LIN {X 0,Y 102.749,Z 789.468,A -85,B 0,C 180,E1 -26714.124,E2 -26714.124} C_VEL
LIN {X 0,Y 103.619,Z 785.992,A -85,B 0,C 180,E1 -26722.206,E2 -26722.206} C_VEL
LIN {X 0,Y 105.515,Z 782.796,A -85,B 0,C 180,E1 -26727.611,E2 -26727.611} C_VEL
LIN {X 0,Y 106.613,Z 781.059,A -85,B 0,C 180,E1 -26730.002,E2 -26730.002} C_VEL
LIN {X 0,Y 107.479,Z 777.383,A -85,B 0,C 180,E1 -26733.751,E2 -26733.751} C_VEL
LIN {X 0,Y 105.034,Z 782.053,A -85,B 0,C 180,E1 -26741.582,E2 -26741.582} C_VEL
LIN {X 0,Y 105.176,Z 785.938,A -85,B 0,C 180,E1 -26750.687,E2 -26750.687} C_VEL
LIN {X 0,Y 107.342,Z 787.959,A -85,B 0,C 180,E1 -26757.28,E2 -26757.28} C_VEL
LIN {X 0,Y 112.126,Z 789.61,A -85,B 0,C 180,E1 -26764.343,E2 -26764.343} C_VEL
LIN {X 0,Y 118.966,Z 790.415,A -85,B 0,C 180,E1 -26770.532,E2 -26770.532} C_VEL
LIN {X 0,Y 127.429,Z 790.46,A -85,B 0,C 180,E1 -26775.808,E2 -26775.808} C_VEL
LIN {X 0,Y 137.179,Z 789.707,A -85,B 0,C 180,E1 -26780.22,E2 -26780.22} C_VEL
LIN {X 0,Y 138.04,Z 789.191,A -85,B 0,C 180,E1 -26781.434,E2 -26781.434} C_VEL
LIN {X 0,Y 129.834,Z 786.499,A -85,B 0,C 180,E1 -26785.251,E2 -26785.251} C_VEL
LIN {X 0,Y 125.752,Z 785.046,A -85,B 0,C 180,E1 -26787.045,E2 -26787.045} C_VEL
LIN {X 0,Y 118.099,Z 782.22,A -85,B 0,C 180,E1 -26789.693,E2 -26789.693} C_VEL
LIN {X 0,Y 110.921,Z 778.802,A -85,B 0,C 180,E1 -26792.656,E2 -26792.656} C_VEL
LIN {X 0,Y 107.697,Z 776.475,A -85,B 0,C 180,E1 -26794.945,E2 -26794.945} C_VEL
LIN {X 0,Y 101.788,Z 769.899,A -85,B 0,C 180,E1 -26801.896,E2 -26801.896} C_VEL
LIN {X 0,Y 97.245,Z 760.94,A -85,B 0,C 180,E1 -26810.64,E2 -26810.64} C_VEL
LIN {X 0,Y 94.988,Z 751.352,A -85,B 0,C 180,E1 -26818.938,E2 -26818.938} C_VEL
LIN {X 0,Y 94.512,Z 741.434,A -85,B 0,C 180,E1 -26826.402,E2 -26826.402} C_VEL
LIN {X 0,Y 94.977,Z 731.323,A -85,B 0,C 180,E1 -26832.824,E2 -26832.824} C_VEL
LIN {X 0,Y 96.352,Z 718.316,A -85,B 0,C 180,E1 -26839.712,E2 -26839.712} C_VEL
LIN {X 0,Y 98.293,Z 705.149,A -85,B 0,C 180,E1 -26845.402,E2 -26845.402} C_VEL
LIN {X 0,Y 100.42,Z 692.066,A -85,B 0,C 180,E1 -26849.909,E2 -26849.909} C_VEL
LIN {X 0,Y 102.876,Z 676.496,A -85,B 0,C 180,E1 -26854.122,E2 -26854.122} C_VEL
LIN {X 0,Y 105.229,Z 659.963,A -85,B 0,C 180,E1 -26857.547,E2 -26857.547} C_VEL
LIN {X 0,Y 106.998,Z 643.946,A -85,B 0,C 180,E1 -26859.974,E2 -26859.974} C_VEL
LIN {X 0,Y 107.849,Z 633.632,A -85,B 0,C 180,E1 -26861.337,E2 -26861.337} C_VEL
LIN {X 0,Y 94.949,Z 593.014,A -85,B 0,C 180,E1 -26868.934,E2 -26868.934} C_VEL
LIN {X 0,Y 93.652,Z 588.813,A -85,B 0,C 180,E1 -26869.886,E2 -26869.886} C_VEL
LIN {X 0,Y 93.6,Z 588.823,A -85,B 0,C 180,E1 -26875.68,E2 -26875.68} C_VEL
LIN {X 0,Y 93.669,Z 588.815,A -85,B 0,C 180,E1 -26884.202,E2 -26884.202} C_VEL
LIN {X 0,Y 93.694,Z 588.809,A -85,B 0,C 180,E1 -26887.97,E2 -26887.97} C_VEL
LIN {X 0,Y 94.097,Z 588.759,A -85,B 0,C 180,E1 -26897.049,E2 -26897.049} C_VEL
LIN {X 0,Y 94.21,Z 588.748,A -85,B 0,C 180,E1 -26901.417,E2 -26901.417} C_VEL
LIN {X 0,Y 94.796,Z 588.676,A -85,B 0,C 180,E1 -26909.997,E2 -26909.997} C_VEL
LIN {X 0,Y 94.212,Z 588.749,A -85,B 0,C 180,E1 -26918.578,E2 -26918.578} C_VEL
LIN {X 0,Y 94.054,Z 588.764,A -85,B 0,C 180,E1 -26923.745,E2 -26923.745} C_VEL
LIN {X 0,Y 93.702,Z 588.806,A -85,B 0,C 180,E1 -26932.023,E2 -26932.023} C_VEL
LIN {X 0,Y 93.623,Z 588.822,A -85,B 0,C 180,E1 -26936.766,E2 -26936.766} C_VEL
LIN {X 0,Y 93.667,Z 588.928,A -85,B 0,C 180,E1 -26939.341,E2 -26939.341} C_VEL
LIN {X 0,Y 101.377,Z 610.141,A -85,B 0,C 180,E1 -26943.866,E2 -26943.866} C_VEL
LIN {X 0,Y 108.869,Z 632.294,A -85,B 0,C 180,E1 -26947.752,E2 -26947.752} C_VEL
LIN {X 0,Y 106.477,Z 660.955,A -85,B 0,C 180,E1 -26951.01,E2 -26951.01} C_VEL
LIN {X 0,Y 104.601,Z 676.009,A -85,B 0,C 180,E1 -26953.411,E2 -26953.411} C_VEL
LIN {X 0,Y 102.104,Z 691.494,A -85,B 0,C 180,E1 -26956.844,E2 -26956.844} C_VEL
LIN {X 0,Y 99.84,Z 704.757,A -85,B 0,C 180,E1 -26960.739,E2 -26960.739} C_VEL
LIN {X 0,Y 97.549,Z 717.311,A -85,B 0,C 180,E1 -26965.436,E2 -26965.436} C_VEL
LIN {X 0,Y 95.603,Z 729.31,A -85,B 0,C 180,E1 -26971.096,E2 -26971.096} C_VEL
LIN {X 0,Y 94.187,Z 741.072,A -85,B 0,C 180,E1 -26978.096,E2 -26978.096} C_VEL
LIN {X 0,Y 93.799,Z 750.604,A -85,B 0,C 180,E1 -26985.021,E2 -26985.021} C_VEL
LIN {X 0,Y 94.678,Z 759.206,A -85,B 0,C 180,E1 -26992.538,E2 -26992.538} C_VEL
LIN {X 0,Y 96.957,Z 766.486,A -85,B 0,C 180,E1 -27000.002,E2 -27000.002} C_VEL
LIN {X 0,Y 101.462,Z 773.182,A -85,B 0,C 180,E1 -27007.965,E2 -27007.965} C_VEL
LIN {X 0,Y 107.752,Z 778.42,A -85,B 0,C 180,E1 -27015.125,E2 -27015.125} C_VEL
LIN {X 0,Y 115.614,Z 782.288,A -85,B 0,C 180,E1 -27021.393,E2 -27021.393} C_VEL
LIN {X 0,Y 124.827,Z 784.879,A -85,B 0,C 180,E1 -27026.772,E2 -27026.772} C_VEL
LIN {X 0,Y 135.125,Z 786.167,A -85,B 0,C 180,E1 -27031.341,E2 -27031.341} C_VEL
LIN {X 0,Y 141.701,Z 786.312,A -85,B 0,C 180,E1 -27033.724,E2 -27033.724} C_VEL
LIN {X 0,Y 140.071,Z 787.038,A -85,B 0,C 180,E1 -27034.847,E2 -27034.847} C_VEL
LIN {X 0,Y 132.441,Z 788.824,A -85,B 0,C 180,E1 -27037.256,E2 -27037.256} C_VEL
LIN {X 0,Y 122.157,Z 790.661,A -85,B 0,C 180,E1 -27041.593,E2 -27041.593} C_VEL
LIN {X 0,Y 113.099,Z 791.524,A -85,B 0,C 180,E1 -27046.882,E2 -27046.882} C_VEL
LIN {X 0,Y 105.583,Z 791.44,A -85,B 0,C 180,E1 -27053.199,E2 -27053.199} C_VEL
LIN {X 0,Y 100.069,Z 790.419,A -85,B 0,C 180,E1 -27060.556,E2 -27060.556} C_VEL
LIN {X 0,Y 96.901,Z 788.403,A -85,B 0,C 180,E1 -27068.74,E2 -27068.74} C_VEL
LIN {X 0,Y 96.617,Z 784.333,A -85,B 0,C 180,E1 -27079.525,E2 -27079.525} C_VEL
LIN {X 0,Y 98.587,Z 780.547,A -85,B 0,C 180,E1 -27086.422,E2 -27086.422} C_VEL
LIN {X 0,Y 100.12,Z 778.059,A -85,B 0,C 180,E1 -27090.002,E2 -27090.002} C_VEL
LIN {X 0,Y 101.197,Z 774.028,A -85,B 0,C 180,E1 -27094.122,E2 -27094.122} C_VEL
LIN {X 0,Y 98.804,Z 778.837,A -85,B 0,C 180,E1 -27102.324,E2 -27102.324} C_VEL
LIN {X 0,Y 98.858,Z 782.558,A -85,B 0,C 180,E1 -27110.824,E2 -27110.824} C_VEL
LIN {X 0,Y 101.494,Z 785.233,A -85,B 0,C 180,E1 -27118.996,E2 -27118.996} C_VEL
LIN {X 0,Y 106.657,Z 787.141,A -85,B 0,C 180,E1 -27126.376,E2 -27126.376} C_VEL
LIN {X 0,Y 113.872,Z 788.266,A -85,B 0,C 180,E1 -27132.761,E2 -27132.761} C_VEL
LIN {X 0,Y 122.734,Z 788.604,A -85,B 0,C 180,E1 -27138.111,E2 -27138.111} C_VEL
LIN {X 0,Y 127.656,Z 788.517,A -85,B 0,C 180,E1 -27140.425,E2 -27140.425} C_VEL
LIN {X 0,Y 128.428,Z 788.232,A -85,B 0,C 180,E1 -27141.286,E2 -27141.286} C_VEL
LIN {X 0,Y 117.182,Z 783.23,A -85,B 0,C 180,E1 -27147.33,E2 -27147.33} C_VEL
LIN {X 0,Y 107.697,Z 776.475,A -85,B 0,C 180,E1 -27154.945,E2 -27154.945} C_VEL
LIN {X 0,Y 104.714,Z 774.045,A -85,B 0,C 180,E1 -27157.328,E2 -27157.328} C_VEL
LIN {X 0,Y 98.763,Z 769.454,A -85,B 0,C 180,E1 -27160.951,E2 -27160.951} C_VEL
LIN {X 0,Y 93.335,Z 764.35,A -85,B 0,C 180,E1 -27164.901,E2 -27164.901} C_VEL
LIN {X 0,Y 91.305,Z 761.124,A -85,B 0,C 180,E1 -27167.749,E2 -27167.749} C_VEL
LIN {X 0,Y 88.506,Z 751.405,A -85,B 0,C 180,E1 -27176.584,E2 -27176.584} C_VEL
LIN {X 0,Y 87.654,Z 741.383,A -85,B 0,C 180,E1 -27184.597,E2 -27184.597} C_VEL
LIN {X 0,Y 87.983,Z 731.28,A -85,B 0,C 180,E1 -27191.517,E2 -27191.517} C_VEL
LIN {X 0,Y 89.131,Z 719.215,A -85,B 0,C 180,E1 -27198.383,E2 -27198.383} C_VEL
LIN {X 0,Y 90.992,Z 706.045,A -85,B 0,C 180,E1 -27204.527,E2 -27204.527} C_VEL
LIN {X 0,Y 93.326,Z 691.502,A -85,B 0,C 180,E1 -27209.925,E2 -27209.925} C_VEL
LIN {X 0,Y 95.591,Z 677.271,A -85,B 0,C 180,E1 -27214.095,E2 -27214.095} C_VEL
LIN {X 0,Y 97.685,Z 663.001,A -85,B 0,C 180,E1 -27217.302,E2 -27217.302} C_VEL
LIN {X 0,Y 99.685,Z 646.899,A -85,B 0,C 180,E1 -27220.01,E2 -27220.01} C_VEL
LIN {X 0,Y 100.723,Z 634.684,A -85,B 0,C 180,E1 -27221.738,E2 -27221.738} C_VEL
LIN {X 0,Y 88.679,Z 596.382,A -85,B 0,C 180,E1 -27229.401,E2 -27229.401} C_VEL
LIN {X 0,Y 86.592,Z 589.696,A -85,B 0,C 180,E1 -27230.991,E2 -27230.991} C_VEL
LIN {X 0,Y 86.546,Z 589.702,A -85,B 0,C 180,E1 -27235.356,E2 -27235.356} C_VEL
LIN {X 0,Y 86.585,Z 589.698,A -85,B 0,C 180,E1 -27243.23,E2 -27243.23} C_VEL
LIN {X 0,Y 86.664,Z 589.69,A -85,B 0,C 180,E1 -27251.069,E2 -27251.069} C_VEL
LIN {X 0,Y 86.968,Z 589.643,A -85,B 0,C 180,E1 -27255.967,E2 -27255.967} C_VEL
LIN {X 0,Y 87.116,Z 589.634,A -85,B 0,C 180,E1 -27260.712,E2 -27260.712} C_VEL
LIN {X 0,Y 87.723,Z 589.557,A -85,B 0,C 180,E1 -27269.997,E2 -27269.997} C_VEL
LIN {X 0,Y 87.12,Z 589.631,A -85,B 0,C 180,E1 -27279.282,E2 -27279.282} C_VEL
LIN {X 0,Y 86.971,Z 589.648,A -85,B 0,C 180,E1 -27284.147,E2 -27284.147} C_VEL
LIN {X 0,Y 86.597,Z 589.697,A -85,B 0,C 180,E1 -27293.937,E2 -27293.937} C_VEL
LIN {X 0,Y 86.582,Z 589.697,A -85,B 0,C 180,E1 -27297.721,E2 -27297.721} C_VEL
LIN {X 0,Y 88.893,Z 595.971,A -85,B 0,C 180,E1 -27299.282,E2 -27299.282} C_VEL
LIN {X 0,Y 95.332,Z 613.924,A -85,B 0,C 180,E1 -27303.247,E2 -27303.247} C_VEL
LIN {X 0,Y 101.871,Z 633.413,A -85,B 0,C 180,E1 -27306.945,E2 -27306.945} C_VEL
LIN {X 0,Y 99.414,Z 661.436,A -85,B 0,C 180,E1 -27310.347,E2 -27310.347} C_VEL
LIN {X 0,Y 97.56,Z 676.097,A -85,B 0,C 180,E1 -27312.79,E2 -27312.79} C_VEL
LIN {X 0,Y 95.145,Z 690.751,A -85,B 0,C 180,E1 -27316.175,E2 -27316.175} C_VEL
LIN {X 0,Y 92.795,Z 704.324,A -85,B 0,C 180,E1 -27320.355,E2 -27320.355} C_VEL
LIN {X 0,Y 90.344,Z 717.603,A -85,B 0,C 180,E1 -27325.67,E2 -27325.67} C_VEL
LIN {X 0,Y 88.3,Z 730.296,A -85,B 0,C 180,E1 -27332.123,E2 -27332.123} C_VEL
LIN {X 0,Y 87.133,Z 740.71,A -85,B 0,C 180,E1 -27338.72,E2 -27338.72} C_VEL
LIN {X 0,Y 86.91,Z 751.311,A -85,B 0,C 180,E1 -27347.03,E2 -27347.03} C_VEL
LIN {X 0,Y 88.236,Z 760.327,A -85,B 0,C 180,E1 -27355.434,E2 -27355.434} C_VEL
LIN {X 0,Y 91.718,Z 768.493,A -85,B 0,C 180,E1 -27364.397,E2 -27364.397} C_VEL
LIN {X 0,Y 97.226,Z 775.055,A -85,B 0,C 180,E1 -27372.526,E2 -27372.526} C_VEL
LIN {X 0,Y 104.578,Z 780.174,A -85,B 0,C 180,E1 -27379.636,E2 -27379.636} C_VEL
LIN {X 0,Y 113.458,Z 783.976,A -85,B 0,C 180,E1 -27385.698,E2 -27385.698} C_VEL
LIN {X 0,Y 123.532,Z 786.488,A -85,B 0,C 180,E1 -27390.801,E2 -27390.801} C_VEL
LIN {X 0,Y 130.09,Z 787.368,A -85,B 0,C 180,E1 -27393.447,E2 -27393.447} C_VEL
LIN {X 0,Y 128.293,Z 787.989,A -85,B 0,C 180,E1 -27394.747,E2 -27394.747} C_VEL
LIN {X 0,Y 117.623,Z 789.414,A -85,B 0,C 180,E1 -27399.039,E2 -27399.039} C_VEL
LIN {X 0,Y 108.116,Z 789.936,A -85,B 0,C 180,E1 -27404.356,E2 -27404.356} C_VEL
LIN {X 0,Y 100.154,Z 789.561,A -85,B 0,C 180,E1 -27410.839,E2 -27410.839} C_VEL
LIN {X 0,Y 94.181,Z 788.241,A -85,B 0,C 180,E1 -27418.513,E2 -27418.513} C_VEL
LIN {X 0,Y 90.644,Z 785.927,A -85,B 0,C 180,E1 -27427.193,E2 -27427.193} C_VEL
LIN {X 0,Y 89.877,Z 782.534,A -85,B 0,C 180,E1 -27436.436,E2 -27436.436} C_VEL
LIN {X 0,Y 91.911,Z 777.889,A -85,B 0,C 180,E1 -27445.617,E2 -27445.617} C_VEL
LIN {X 0,Y 93.702,Z 774.893,A -85,B 0,C 180,E1 -27450.003,E2 -27450.003} C_VEL
LIN {X 0,Y 94.986,Z 770.578,A -85,B 0,C 180,E1 -27454.538,E2 -27454.538} C_VEL
LIN {X 0,Y 92.654,Z 775.486,A -85,B 0,C 180,E1 -27463.156,E2 -27463.156} C_VEL
LIN {X 0,Y 92.865,Z 779.416,A -85,B 0,C 180,E1 -27472.237,E2 -27472.237} C_VEL
LIN {X 0,Y 95.808,Z 782.382,A -85,B 0,C 180,E1 -27480.899,E2 -27480.899} C_VEL
LIN {X 0,Y 101.388,Z 784.532,A -85,B 0,C 180,E1 -27488.602,E2 -27488.602} C_VEL
LIN {X 0,Y 109.024,Z 785.949,A -85,B 0,C 180,E1 -27495.164,E2 -27495.164} C_VEL
LIN {X 0,Y 118.28,Z 786.587,A -85,B 0,C 180,E1 -27500.576,E2 -27500.576} C_VEL
LIN {X 0,Y 115.862,Z 785.109,A -85,B 0,C 180,E1 -27502.655,E2 -27502.655} C_VEL
LIN {X 0,Y 107.045,Z 779.918,A -85,B 0,C 180,E1 -27508.314,E2 -27508.314} C_VEL
LIN {X 0,Y 99.692,Z 773.713,A -85,B 0,C 180,E1 -27514.975,E2 -27514.975} C_VEL
LIN {X 0,Y 93.336,Z 765.345,A -85,B 0,C 180,E1 -27523.597,E2 -27523.597} C_VEL
LIN {X 0,Y 91.305,Z 761.124,A -85,B 0,C 180,E1 -27527.749,E2 -27527.749} C_VEL
LIN {X 0,Y 89.543,Z 757.815,A -85,B 0,C 180,E1 -27530.63,E2 -27530.63} C_VEL
LIN {X 0,Y 85.483,Z 751.733,A -85,B 0,C 180,E1 -27535.013,E2 -27535.013} C_VEL
LIN {X 0,Y 81.885,Z 745.179,A -85,B 0,C 180,E1 -27539.55,E2 -27539.55} C_VEL
LIN {X 0,Y 80.958,Z 741.128,A -85,B 0,C 180,E1 -27542.552,E2 -27542.552} C_VEL
LIN {X 0,Y 81.054,Z 731.038,A -85,B 0,C 180,E1 -27549.984,E2 -27549.984} C_VEL
LIN {X 0,Y 82.123,Z 718.467,A -85,B 0,C 180,E1 -27557.681,E2 -27557.681} C_VEL
LIN {X 0,Y 83.917,Z 705.56,A -85,B 0,C 180,E1 -27564.094,E2 -27564.094} C_VEL
LIN {X 0,Y 86.268,Z 690.738,A -85,B 0,C 180,E1 -27569.93,E2 -27569.93} C_VEL
LIN {X 0,Y 88.61,Z 676.201,A -85,B 0,C 180,E1 -27574.408,E2 -27574.408} C_VEL
LIN {X 0,Y 90.788,Z 661.359,A -85,B 0,C 180,E1 -27577.91,E2 -27577.91} C_VEL
LIN {X 0,Y 92.945,Z 643.781,A -85,B 0,C 180,E1 -27580.974,E2 -27580.974} C_VEL
LIN {X 0,Y 93.679,Z 635.932,A -85,B 0,C 180,E1 -27582.193,E2 -27582.193} C_VEL
LIN {X 0,Y 81.692,Z 597.606,A -85,B 0,C 180,E1 -27590.416,E2 -27590.416} C_VEL
LIN {X 0,Y 79.502,Z 590.581,A -85,B 0,C 180,E1 -27592.358,E2 -27592.358} C_VEL
LIN {X 0,Y 79.483,Z 590.584,A -85,B 0,C 180,E1 -27602.15,E2 -27602.15} C_VEL
LIN {X 0,Y 79.523,Z 590.578,A -85,B 0,C 180,E1 -27609.295,E2 -27609.295} C_VEL
LIN {X 0,Y 79.84,Z 590.531,A -85,B 0,C 180,E1 -27615.522,E2 -27615.522} C_VEL
LIN {X 0,Y 79.999,Z 590.52,A -85,B 0,C 180,E1 -27619.877,E2 -27619.877} C_VEL
LIN {X 0,Y 80.651,Z 590.438,A -85,B 0,C 180,E1 -27629.997,E2 -27629.997} C_VEL
LIN {X 0,Y 80.001,Z 590.516,A -85,B 0,C 180,E1 -27640.116,E2 -27640.116} C_VEL
LIN {X 0,Y 79.812,Z 590.542,A -85,B 0,C 180,E1 -27645.315,E2 -27645.315} C_VEL
LIN {X 0,Y 79.567,Z 590.727,A -85,B 0,C 180,E1 -27655.853,E2 -27655.853} C_VEL
LIN {X 0,Y 86.204,Z 608.745,A -85,B 0,C 180,E1 -27660.628,E2 -27660.628} C_VEL
LIN {X 0,Y 94.91,Z 634.731,A -85,B 0,C 180,E1 -27666.077,E2 -27666.077} C_VEL
LIN {X 0,Y 92.379,Z 662.051,A -85,B 0,C 180,E1 -27669.639,E2 -27669.639} C_VEL
LIN {X 0,Y 90.346,Z 677.161,A -85,B 0,C 180,E1 -27672.356,E2 -27672.356} C_VEL
LIN {X 0,Y 87.873,Z 691.767,A -85,B 0,C 180,E1 -27676.034,E2 -27676.034} C_VEL
LIN {X 0,Y 85.505,Z 704.995,A -85,B 0,C 180,E1 -27680.434,E2 -27680.434} C_VEL
LIN {X 0,Y 83.052,Z 718.213,A -85,B 0,C 180,E1 -27686.123,E2 -27686.123} C_VEL
LIN {X 0,Y 81.251,Z 729.47,A -85,B 0,C 180,E1 -27692.297,E2 -27692.297} C_VEL
LIN {X 0,Y 80.114,Z 740.071,A -85,B 0,C 180,E1 -27699.46,E2 -27699.46} C_VEL
LIN {X 0,Y 79.968,Z 750.161,A -85,B 0,C 180,E1 -27707.694,E2 -27707.694} C_VEL
LIN {X 0,Y 81.35,Z 758.973,A -85,B 0,C 180,E1 -27716.287,E2 -27716.287} C_VEL
LIN {X 0,Y 84.677,Z 766.993,A -85,B 0,C 180,E1 -27725.174,E2 -27725.174} C_VEL
LIN {X 0,Y 90.124,Z 773.814,A -85,B 0,C 180,E1 -27733.532,E2 -27733.532} C_VEL
LIN {X 0,Y 98.121,Z 779.792,A -85,B 0,C 180,E1 -27741.395,E2 -27741.395} C_VEL
LIN {X 0,Y 106.891,Z 783.919,A -85,B 0,C 180,E1 -27747.405,E2 -27747.405} C_VEL
LIN {X 0,Y 117.289,Z 787.007,A -85,B 0,C 180,E1 -27752.637,E2 -27752.637} C_VEL
LIN {X 0,Y 118.743,Z 787.604,A -85,B 0,C 180,E1 -27754.047,E2 -27754.047} C_VEL
LIN {X 0,Y 108.211,Z 788.237,A -85,B 0,C 180,E1 -27758.801,E2 -27758.801} C_VEL
LIN {X 0,Y 98.955,Z 788,A -85,B 0,C 180,E1 -27764.751,E2 -27764.751} C_VEL
LIN {X 0,Y 91.39,Z 786.844,A -85,B 0,C 180,E1 -27772.036,E2 -27772.036} C_VEL
LIN {X 0,Y 86.154,Z 784.735,A -85,B 0,C 180,E1 -27780.699,E2 -27780.699} C_VEL
LIN {X 0,Y 83.665,Z 781.621,A -85,B 0,C 180,E1 -27790.369,E2 -27790.369} C_VEL
LIN {X 0,Y 84.181,Z 777.375,A -85,B 0,C 180,E1 -27800.391,E2 -27800.391} C_VEL
LIN {X 0,Y 86.446,Z 773.3,A -85,B 0,C 180,E1 -27807.673,E2 -27807.673} C_VEL
LIN {X 0,Y 87.331,Z 771.63,A -85,B 0,C 180,E1 -27810.003,E2 -27810.003} C_VEL
LIN {X 0,Y 88.862,Z 766.986,A -85,B 0,C 180,E1 -27815.026,E2 -27815.026} C_VEL
LIN {X 0,Y 86.595,Z 772.016,A -85,B 0,C 180,E1 -27824.095,E2 -27824.095} C_VEL
LIN {X 0,Y 87.004,Z 776.136,A -85,B 0,C 180,E1 -27833.825,E2 -27833.825} C_VEL
LIN {X 0,Y 90.325,Z 779.351,A -85,B 0,C 180,E1 -27843.004,E2 -27843.004} C_VEL
LIN {X 0,Y 96.336,Z 781.777,A -85,B 0,C 180,E1 -27851.043,E2 -27851.043} C_VEL
LIN {X 0,Y 104.431,Z 783.447,A -85,B 0,C 180,E1 -27857.758,E2 -27857.758} C_VEL
LIN {X 0,Y 109.092,Z 784.025,A -85,B 0,C 180,E1 -27860.634,E2 -27860.634} C_VEL
LIN {X 0,Y 105.528,Z 781.783,A -85,B 0,C 180,E1 -27863.172,E2 -27863.172} C_VEL
LIN {X 0,Y 97.051,Z 775.666,A -85,B 0,C 180,E1 -27869.54,E2 -27869.54} C_VEL
LIN {X 0,Y 90.105,Z 768.449,A -85,B 0,C 180,E1 -27877.044,E2 -27877.044} C_VEL
LIN {X 0,Y 84.587,Z 758.828,A -85,B 0,C 180,E1 -27886.79,E2 -27886.79} C_VEL
LIN {X 0,Y 81.681,Z 748.575,A -85,B 0,C 180,E1 -27896.298,E2 -27896.298} C_VEL
LIN {X 0,Y 80.958,Z 741.128,A -85,B 0,C 180,E1 -27902.552,E2 -27902.552} C_VEL
LIN {X 0,Y 80.216,Z 737.053,A -85,B 0,C 180,E1 -27905.46,E2 -27905.46} C_VEL
LIN {X 0,Y 77.637,Z 729.704,A -85,B 0,C 180,E1 -27909.868,E2 -27909.868} C_VEL
LIN {X 0,Y 75.366,Z 721.87,A -85,B 0,C 180,E1 -27914.286,E2 -27914.286} C_VEL
LIN {X 0,Y 75.215,Z 717.068,A -85,B 0,C 180,E1 -27917.071,E2 -27917.071} C_VEL
LIN {X 0,Y 77.032,Z 703.675,A -85,B 0,C 180,E1 -27924.162,E2 -27924.162} C_VEL
LIN {X 0,Y 79.215,Z 689.969,A -85,B 0,C 180,E1 -27929.935,E2 -27929.935} C_VEL
LIN {X 0,Y 81.653,Z 674.969,A -85,B 0,C 180,E1 -27934.763,E2 -27934.763} C_VEL
LIN {X 0,Y 84.123,Z 658.297,A -85,B 0,C 180,E1 -27938.796,E2 -27938.796} C_VEL
LIN {X 0,Y 86.483,Z 637.7,A -85,B 0,C 180,E1 -27942.435,E2 -27942.435} C_VEL
LIN {X 0,Y 86.192,Z 635.836,A -85,B 0,C 180,E1 -27942.786,E2 -27942.786} C_VEL
LIN {X 0,Y 75.123,Z 600.002,A -85,B 0,C 180,E1 -27951.31,E2 -27951.31} C_VEL
LIN {X 0,Y 72.375,Z 591.47,A -85,B 0,C 180,E1 -27953.835,E2 -27953.835} C_VEL
LIN {X 0,Y 72.392,Z 591.467,A -85,B 0,C 180,E1 -27960.957,E2 -27960.957} C_VEL
LIN {X 0,Y 72.399,Z 591.458,A -85,B 0,C 180,E1 -27967.148,E2 -27967.148} C_VEL
LIN {X 0,Y 72.756,Z 591.413,A -85,B 0,C 180,E1 -27974.999,E2 -27974.999} C_VEL
LIN {X 0,Y 72.883,Z 591.406,A -85,B 0,C 180,E1 -27978.877,E2 -27978.877} C_VEL
LIN {X 0,Y 73.578,Z 591.319,A -85,B 0,C 180,E1 -27989.997,E2 -27989.997} C_VEL
LIN {X 0,Y 72.894,Z 591.396,A -85,B 0,C 180,E1 -28001.115,E2 -28001.115} C_VEL
LIN {X 0,Y 72.608,Z 591.441,A -85,B 0,C 180,E1 -28006.877,E2 -28006.877} C_VEL
LIN {X 0,Y 72.523,Z 591.569,A -85,B 0,C 180,E1 -28013.748,E2 -28013.748} C_VEL
LIN {X 0,Y 79.037,Z 609.073,A -85,B 0,C 180,E1 -28018.897,E2 -28018.897} C_VEL
LIN {X 0,Y 86.705,Z 632.084,A -85,B 0,C 180,E1 -28024.348,E2 -28024.348} C_VEL
LIN {X 0,Y 87.955,Z 635.908,A -85,B 0,C 180,E1 -28025.146,E2 -28025.146} C_VEL
LIN {X 0,Y 85.273,Z 662.842,A -85,B 0,C 180,E1 -28028.942,E2 -28028.942} C_VEL
LIN {X 0,Y 83.198,Z 677.671,A -85,B 0,C 180,E1 -28031.792,E2 -28031.792} C_VEL
LIN {X 0,Y 80.818,Z 691.48,A -85,B 0,C 180,E1 -28035.464,E2 -28035.464} C_VEL
LIN {X 0,Y 78.353,Z 704.949,A -85,B 0,C 180,E1 -28040.279,E2 -28040.279} C_VEL
LIN {X 0,Y 75.93,Z 717.835,A -85,B 0,C 180,E1 -28046.268,E2 -28046.268} C_VEL
LIN {X 0,Y 74.077,Z 729.559,A -85,B 0,C 180,E1 -28053.217,E2 -28053.217} C_VEL
LIN {X 0,Y 73.005,Z 741.127,A -85,B 0,C 180,E1 -28061.77,E2 -28061.77} C_VEL
LIN {X 0,Y 73.263,Z 750.638,A -85,B 0,C 180,E1 -28070.338,E2 -28070.338} C_VEL
LIN {X 0,Y 75.29,Z 759.932,A -85,B 0,C 180,E1 -28080.002,E2 -28080.002} C_VEL
LIN {X 0,Y 79.912,Z 768.551,A -85,B 0,C 180,E1 -28090.133,E2 -28090.133} C_VEL
LIN {X 0,Y 86.786,Z 775.619,A -85,B 0,C 180,E1 -28098.903,E2 -28098.903} C_VEL
LIN {X 0,Y 95.504,Z 781.25,A -85,B 0,C 180,E1 -28106.204,E2 -28106.204} C_VEL
LIN {X 0,Y 105.695,Z 785.553,A -85,B 0,C 180,E1 -28112.139,E2 -28112.139} C_VEL
LIN {X 0,Y 108.165,Z 786.328,A -85,B 0,C 180,E1 -28113.324,E2 -28113.324} C_VEL
LIN {X 0,Y 107.168,Z 786.544,A -85,B 0,C 180,E1 -28114.323,E2 -28114.323} C_VEL
LIN {X 0,Y 98.958,Z 786.38,A -85,B 0,C 180,E1 -28118.632,E2 -28118.632} C_VEL
LIN {X 0,Y 89.98,Z 785.347,A -85,B 0,C 180,E1 -28125.339,E2 -28125.339} C_VEL
LIN {X 0,Y 82.964,Z 783.426,A -85,B 0,C 180,E1 -28133.635,E2 -28133.635} C_VEL
LIN {X 0,Y 78.576,Z 780.553,A -85,B 0,C 180,E1 -28143.439,E2 -28143.439} C_VEL
LIN {X 0,Y 77.266,Z 776.621,A -85,B 0,C 180,E1 -28154.168,E2 -28154.168} C_VEL
LIN {X 0,Y 79.232,Z 771.463,A -85,B 0,C 180,E1 -28164.914,E2 -28164.914} C_VEL
LIN {X 0,Y 81.047,Z 768.182,A -85,B 0,C 180,E1 -28170.003,E2 -28170.003} C_VEL
LIN {X 0,Y 82.845,Z 763.293,A -85,B 0,C 180,E1 -28175.632,E2 -28175.632} C_VEL
LIN {X 0,Y 80.589,Z 768.93,A -85,B 0,C 180,E1 -28186.398,E2 -28186.398} C_VEL
LIN {X 0,Y 81.294,Z 772.742,A -85,B 0,C 180,E1 -28195.614,E2 -28195.614} C_VEL
LIN {X 0,Y 85.044,Z 776.154,A -85,B 0,C 180,E1 -28205.347,E2 -28205.347} C_VEL
LIN {X 0,Y 91.518,Z 778.865,A -85,B 0,C 180,E1 -28213.724,E2 -28213.724} C_VEL
LIN {X 0,Y 100.114,Z 780.783,A -85,B 0,C 180,E1 -28220.555,E2 -28220.555} C_VEL
LIN {X 0,Y 91.095,Z 774.106,A -85,B 0,C 180,E1 -28227.311,E2 -28227.311} C_VEL
LIN {X 0,Y 83.004,Z 765.383,A -85,B 0,C 180,E1 -28236.283,E2 -28236.283} C_VEL
LIN {X 0,Y 77.453,Z 754.997,A -85,B 0,C 180,E1 -28246.886,E2 -28246.886} C_VEL
LIN {X 0,Y 74.753,Z 743.955,A -85,B 0,C 180,E1 -28257.303,E2 -28257.303} C_VEL
LIN {X 0,Y 74.192,Z 732.439,A -85,B 0,C 180,E1 -28266.798,E2 -28266.798} C_VEL
LIN {X 0,Y 74.822,Z 720.543,A -85,B 0,C 180,E1 -28274.967,E2 -28274.967} C_VEL
LIN {X 0,Y 75.215,Z 717.068,A -85,B 0,C 180,E1 -28277.071,E2 -28277.071} C_VEL
LIN {X 0,Y 75.166,Z 712.273,A -85,B 0,C 180,E1 -28279.687,E2 -28279.687} C_VEL
LIN {X 0,Y 73.492,Z 703.913,A -85,B 0,C 180,E1 -28283.58,E2 -28283.58} C_VEL
LIN {X 0,Y 71.911,Z 695.224,A -85,B 0,C 180,E1 -28287.284,E2 -28287.284} C_VEL
LIN {X 0,Y 72.059,Z 689.914,A -85,B 0,C 180,E1 -28289.444,E2 -28289.444} C_VEL
LIN {X 0,Y 74.535,Z 674.577,A -85,B 0,C 180,E1 -28294.862,E2 -28294.862} C_VEL
LIN {X 0,Y 76.88,Z 659.18,A -85,B 0,C 180,E1 -28298.935,E2 -28298.935} C_VEL
LIN {X 0,Y 79.381,Z 638.425,A -85,B 0,C 180,E1 -28302.918,E2 -28302.918} C_VEL
LIN {X 0,Y 75.687,Z 625.888,A -85,B 0,C 180,E1 -28305.855,E2 -28305.855} C_VEL
LIN {X 0,Y 67.223,Z 598.131,A -85,B 0,C 180,E1 -28313.51,E2 -28313.51} C_VEL
LIN {X 0,Y 65.249,Z 592.352,A -85,B 0,C 180,E1 -28315.56,E2 -28315.56} C_VEL
LIN {X 0,Y 65.249,Z 592.352,A -85,B 0,C 180,E1 -28324.475,E2 -28324.475} C_VEL
LIN {X 0,Y 65.65,Z 592.299,A -85,B 0,C 180,E1 -28334.455,E2 -28334.455} C_VEL
LIN {X 0,Y 65.782,Z 592.287,A -85,B 0,C 180,E1 -28337.659,E2 -28337.659} C_VEL
LIN {X 0,Y 66.502,Z 592.2,A -85,B 0,C 180,E1 -28349.996,E2 -28349.996} C_VEL
LIN {X 0,Y 65.796,Z 592.279,A -85,B 0,C 180,E1 -28362.331,E2 -28362.331} C_VEL
LIN {X 0,Y 65.408,Z 592.328,A -85,B 0,C 180,E1 -28371.052,E2 -28371.052} C_VEL
LIN {X 0,Y 66.426,Z 595.198,A -85,B 0,C 180,E1 -28372.139,E2 -28372.139} C_VEL
LIN {X 0,Y 71.783,Z 609.089,A -85,B 0,C 180,E1 -28376.901,E2 -28376.901} C_VEL
LIN {X 0,Y 79.471,Z 632.409,A -85,B 0,C 180,E1 -28383.002,E2 -28383.002} C_VEL
LIN {X 0,Y 80.991,Z 637.326,A -85,B 0,C 180,E1 -28384.133,E2 -28384.133} C_VEL
LIN {X 0,Y 78.063,Z 664.816,A -85,B 0,C 180,E1 -28388.356,E2 -28388.356} C_VEL
LIN {X 0,Y 75.953,Z 678.71,A -85,B 0,C 180,E1 -28391.318,E2 -28391.318} C_VEL
LIN {X 0,Y 73.593,Z 692.084,A -85,B 0,C 180,E1 -28395.23,E2 -28395.23} C_VEL
LIN {X 0,Y 70.919,Z 706.249,A -85,B 0,C 180,E1 -28400.824,E2 -28400.824} C_VEL
LIN {X 0,Y 68.433,Z 719.64,A -85,B 0,C 180,E1 -28407.782,E2 -28407.782} C_VEL
LIN {X 0,Y 66.801,Z 730.581,A -85,B 0,C 180,E1 -28415.116,E2 -28415.116} C_VEL
LIN {X 0,Y 66.112,Z 740.339,A -85,B 0,C 180,E1 -28423.072,E2 -28423.072} C_VEL
LIN {X 0,Y 66.571,Z 750.029,A -85,B 0,C 180,E1 -28432.42,E2 -28432.42} C_VEL
LIN {X 0,Y 69.083,Z 759.475,A -85,B 0,C 180,E1 -28442.918,E2 -28442.918} C_VEL
LIN {X 0,Y 74.417,Z 768.464,A -85,B 0,C 180,E1 -28453.659,E2 -28453.659} C_VEL
LIN {X 0,Y 82.054,Z 775.721,A -85,B 0,C 180,E1 -28462.673,E2 -28462.673} C_VEL
LIN {X 0,Y 91.513,Z 781.596,A -85,B 0,C 180,E1 -28469.948,E2 -28469.948} C_VEL
LIN {X 0,Y 97.306,Z 784.262,A -85,B 0,C 180,E1 -28473.271,E2 -28473.271} C_VEL
LIN {X 0,Y 96.204,Z 784.449,A -85,B 0,C 180,E1 -28474.642,E2 -28474.642} C_VEL
LIN {X 0,Y 85.311,Z 783.005,A -85,B 0,C 180,E1 -28482.151,E2 -28482.151} C_VEL
LIN {X 0,Y 77.716,Z 780.789,A -85,B 0,C 180,E1 -28490.731,E2 -28490.731} C_VEL
LIN {X 0,Y 72.77,Z 777.651,A -85,B 0,C 180,E1 -28501.13,E2 -28501.13} C_VEL
LIN {X 0,Y 71.12,Z 773.485,A -85,B 0,C 180,E1 -28512.759,E2 -28512.759} C_VEL
LIN {X 0,Y 73.002,Z 768.081,A -85,B 0,C 180,E1 -28524.479,E2 -28524.479} C_VEL
LIN {X 0,Y 73.995,Z 766.467,A -85,B 0,C 180,E1 -28527.281,E2 -28527.281} C_VEL
LIN {X 0,Y 75.142,Z 763.451,A -85,B 0,C 180,E1 -28531.343,E2 -28531.343} C_VEL
LIN {X 0,Y 76.967,Z 759.413,A -85,B 0,C 180,E1 -28536.228,E2 -28536.228} C_VEL
LIN {X 0,Y 74.86,Z 764.569,A -85,B 0,C 180,E1 -28546.362,E2 -28546.362} C_VEL
LIN {X 0,Y 75.766,Z 769.154,A -85,B 0,C 180,E1 -28557.636,E2 -28557.636} C_VEL
LIN {X 0,Y 79.978,Z 772.825,A -85,B 0,C 180,E1 -28567.964,E2 -28567.964} C_VEL
LIN {X 0,Y 89.057,Z 776.363,A -85,B 0,C 180,E1 -28578.463,E2 -28578.463} C_VEL
LIN {X 0,Y 90.12,Z 776.66,A -85,B 0,C 180,E1 -28579.341,E2 -28579.341} C_VEL
LIN {X 0,Y 90.838,Z 776.642,A -85,B 0,C 180,E1 -28580.544,E2 -28580.544} C_VEL
LIN {X 0,Y 80.318,Z 767.301,A -85,B 0,C 180,E1 -28589.789,E2 -28589.789} C_VEL
LIN {X 0,Y 73.179,Z 757.149,A -85,B 0,C 180,E1 -28600.356,E2 -28600.356} C_VEL
LIN {X 0,Y 69.176,Z 746.447,A -85,B 0,C 180,E1 -28611.232,E2 -28611.232} C_VEL
LIN {X 0,Y 67.634,Z 735.367,A -85,B 0,C 180,E1 -28621.486,E2 -28621.486} C_VEL
LIN {X 0,Y 67.695,Z 724.076,A -85,B 0,C 180,E1 -28630.465,E2 -28630.465} C_VEL
LIN {X 0,Y 68.784,Z 711.744,A -85,B 0,C 180,E1 -28638.608,E2 -28638.608} C_VEL
LIN {X 0,Y 70.71,Z 698.115,A -85,B 0,C 180,E1 -28645.882,E2 -28645.882} C_VEL
LIN {X 0,Y 72.059,Z 689.914,A -85,B 0,C 180,E1 -28649.444,E2 -28649.444} C_VEL
LIN {X 0,Y 72.238,Z 684.671,A -85,B 0,C 180,E1 -28651.445,E2 -28651.445} C_VEL
LIN {X 0,Y 70.862,Z 675.625,A -85,B 0,C 180,E1 -28654.464,E2 -28654.464} C_VEL
LIN {X 0,Y 69.414,Z 666.32,A -85,B 0,C 180,E1 -28657.277,E2 -28657.277} C_VEL
LIN {X 0,Y 69.514,Z 660.614,A -85,B 0,C 180,E1 -28658.796,E2 -28658.796} C_VEL
LIN {X 0,Y 72.229,Z 639.184,A -85,B 0,C 180,E1 -28663.433,E2 -28663.433} C_VEL
LIN {X 0,Y 67.438,Z 623.118,A -85,B 0,C 180,E1 -28667.609,E2 -28667.609} C_VEL
LIN {X 0,Y 60.48,Z 600.063,A -85,B 0,C 180,E1 -28674.808,E2 -28674.808} C_VEL
LIN {X 0,Y 58.184,Z 593.227,A -85,B 0,C 180,E1 -28677.514,E2 -28677.514} C_VEL
LIN {X 0,Y 58.153,Z 593.24,A -85,B 0,C 180,E1 -28681.087,E2 -28681.087} C_VEL
LIN {X 0,Y 58.536,Z 593.186,A -85,B 0,C 180,E1 -28693.83,E2 -28693.83} C_VEL
LIN {X 0,Y 58.822,Z 593.149,A -85,B 0,C 180,E1 -28703.134,E2 -28703.134} C_VEL
LIN {X 0,Y 59.395,Z 593.086,A -85,B 0,C 180,E1 -28709.996,E2 -28709.996} C_VEL
LIN {X 0,Y 58.828,Z 593.157,A -85,B 0,C 180,E1 -28716.857,E2 -28716.857} C_VEL
LIN {X 0,Y 58.55,Z 593.192,A -85,B 0,C 180,E1 -28726.217,E2 -28726.217} C_VEL
LIN {X 0,Y 58.419,Z 593.206,A -85,B 0,C 180,E1 -28728.004,E2 -28728.004} C_VEL
LIN {X 0,Y 60.161,Z 597.993,A -85,B 0,C 180,E1 -28730.123,E2 -28730.123} C_VEL
LIN {X 0,Y 64.755,Z 609.748,A -85,B 0,C 180,E1 -28734.652,E2 -28734.652} C_VEL
LIN {X 0,Y 70.912,Z 628.609,A -85,B 0,C 180,E1 -28740.419,E2 -28740.419} C_VEL
LIN {X 0,Y 73.971,Z 638.132,A -85,B 0,C 180,E1 -28742.907,E2 -28742.907} C_VEL
LIN {X 0,Y 71.266,Z 663.236,A -85,B 0,C 180,E1 -28747.105,E2 -28747.105} C_VEL
LIN {X 0,Y 69.075,Z 677.585,A -85,B 0,C 180,E1 -28750.267,E2 -28750.267} C_VEL
LIN {X 0,Y 66.378,Z 692.52,A -85,B 0,C 180,E1 -28754.927,E2 -28754.927} C_VEL
LIN {X 0,Y 63.943,Z 705.081,A -85,B 0,C 180,E1 -28760.292,E2 -28760.292} C_VEL
LIN {X 0,Y 61.416,Z 718.711,A -85,B 0,C 180,E1 -28768.049,E2 -28768.049} C_VEL
LIN {X 0,Y 59.787,Z 730.437,A -85,B 0,C 180,E1 -28776.629,E2 -28776.629} C_VEL
LIN {X 0,Y 59.245,Z 741.074,A -85,B 0,C 180,E1 -28786.279,E2 -28786.279} C_VEL
LIN {X 0,Y 60.357,Z 750.74,A -85,B 0,C 180,E1 -28796.665,E2 -28796.665} C_VEL
LIN {X 0,Y 63.929,Z 760.584,A -85,B 0,C 180,E1 -28808.375,E2 -28808.375} C_VEL
LIN {X 0,Y 70.189,Z 769.173,A -85,B 0,C 180,E1 -28818.994,E2 -28818.994} C_VEL
LIN {X 0,Y 77.729,Z 775.72,A -85,B 0,C 180,E1 -28826.88,E2 -28826.88} C_VEL
LIN {X 0,Y 86.583,Z 781.165,A -85,B 0,C 180,E1 -28833.225,E2 -28833.225} C_VEL
LIN {X 0,Y 86.182,Z 781.514,A -85,B 0,C 180,E1 -28834.811,E2 -28834.811} C_VEL
LIN {X 0,Y 76.551,Z 779.386,A -85,B 0,C 180,E1 -28842.743,E2 -28842.743} C_VEL
LIN {X 0,Y 69.557,Z 776.447,A -85,B 0,C 180,E1 -28852.687,E2 -28852.687} C_VEL
LIN {X 0,Y 65.699,Z 772.547,A -85,B 0,C 180,E1 -28864.67,E2 -28864.67} C_VEL
LIN {X 0,Y 65.544,Z 767.525,A -85,B 0,C 180,E1 -28877.62,E2 -28877.62} C_VEL
LIN {X 0,Y 67.899,Z 762.861,A -85,B 0,C 180,E1 -28887.037,E2 -28887.037} C_VEL
LIN {X 0,Y 69.052,Z 759.656,A -85,B 0,C 180,E1 -28891.461,E2 -28891.461} C_VEL
LIN {X 0,Y 71.234,Z 755.307,A -85,B 0,C 180,E1 -28896.731,E2 -28896.731} C_VEL
LIN {X 0,Y 69.2,Z 760.615,A -85,B 0,C 180,E1 -28907.742,E2 -28907.742} C_VEL
LIN {X 0,Y 70.437,Z 765.414,A -85,B 0,C 180,E1 -28919.93,E2 -28919.93} C_VEL
LIN {X 0,Y 76.238,Z 769.883,A -85,B 0,C 180,E1 -28932.48,E2 -28932.48} C_VEL
LIN {X 0,Y 81.555,Z 772.078,A -85,B 0,C 180,E1 -28938.699,E2 -28938.699} C_VEL
LIN {X 0,Y 82.119,Z 772.011,A -85,B 0,C 180,E1 -28940.11,E2 -28940.11} C_VEL
LIN {X 0,Y 72.561,Z 762.596,A -85,B 0,C 180,E1 -28949.434,E2 -28949.434} C_VEL
LIN {X 0,Y 66.262,Z 752.828,A -85,B 0,C 180,E1 -28959.833,E2 -28959.833} C_VEL
LIN {X 0,Y 62.616,Z 742.803,A -85,B 0,C 180,E1 -28970.305,E2 -28970.305} C_VEL
LIN {X 0,Y 61.156,Z 732.865,A -85,B 0,C 180,E1 -28979.997,E2 -28979.997} C_VEL
LIN {X 0,Y 61.012,Z 722.209,A -85,B 0,C 180,E1 -28989.11,E2 -28989.11} C_VEL
LIN {X 0,Y 62.025,Z 709.483,A -85,B 0,C 180,E1 -28998.153,E2 -28998.153} C_VEL
LIN {X 0,Y 63.718,Z 697.048,A -85,B 0,C 180,E1 -29005.3,E2 -29005.3} C_VEL
LIN {X 0,Y 65.926,Z 683.424,A -85,B 0,C 180,E1 -29011.472,E2 -29011.472} C_VEL
LIN {X 0,Y 68.344,Z 668.298,A -85,B 0,C 180,E1 -29016.703,E2 -29016.703} C_VEL
LIN {X 0,Y 69.514,Z 660.614,A -85,B 0,C 180,E1 -29018.796,E2 -29018.796} C_VEL
LIN {X 0,Y 69.509,Z 654.938,A -85,B 0,C 180,E1 -29020.172,E2 -29020.172} C_VEL
LIN {X 0,Y 68.434,Z 649.315,A -85,B 0,C 180,E1 -29021.528,E2 -29021.528} C_VEL
LIN {X 0,Y 62.399,Z 630.842,A -85,B 0,C 180,E1 -29026.455,E2 -29026.455} C_VEL
LIN {X 0,Y 54.154,Z 603.146,A -85,B 0,C 180,E1 -29035.857,E2 -29035.857} C_VEL
LIN {X 0,Y 51.118,Z 594.112,A -85,B 0,C 180,E1 -29039.959,E2 -29039.959} C_VEL
LIN {X 0,Y 51.481,Z 594.063,A -85,B 0,C 180,E1 -29054.15,E2 -29054.15} C_VEL
LIN {X 0,Y 51.698,Z 594.039,A -85,B 0,C 180,E1 -29062.182,E2 -29062.182} C_VEL
LIN {X 0,Y 52.28,Z 593.971,A -85,B 0,C 180,E1 -29069.995,E2 -29069.995} C_VEL
LIN {X 0,Y 51.621,Z 594.159,A -85,B 0,C 180,E1 -29084.281,E2 -29084.281} C_VEL
LIN {X 0,Y 53.424,Z 599.261,A -85,B 0,C 180,E1 -29086.881,E2 -29086.881} C_VEL
LIN {X 0,Y 57.157,Z 608.863,A -85,B 0,C 180,E1 -29091.411,E2 -29091.411} C_VEL
LIN {X 0,Y 61.828,Z 622.683,A -85,B 0,C 180,E1 -29096.527,E2 -29096.527} C_VEL
LIN {X 0,Y 67.04,Z 639.439,A -85,B 0,C 180,E1 -29101.608,E2 -29101.608} C_VEL
LIN {X 0,Y 64.151,Z 664.084,A -85,B 0,C 180,E1 -29106.107,E2 -29106.107} C_VEL
LIN {X 0,Y 61.956,Z 677.692,A -85,B 0,C 180,E1 -29109.401,E2 -29109.401} C_VEL
LIN {X 0,Y 59.197,Z 692.614,A -85,B 0,C 180,E1 -29114.58,E2 -29114.58} C_VEL
LIN {X 0,Y 56.745,Z 704.94,A -85,B 0,C 180,E1 -29120.408,E2 -29120.408} C_VEL
LIN {X 0,Y 54.286,Z 718.278,A -85,B 0,C 180,E1 -29128.816,E2 -29128.816} C_VEL
LIN {X 0,Y 52.876,Z 729.161,A -85,B 0,C 180,E1 -29137.682,E2 -29137.682} C_VEL
LIN {X 0,Y 52.57,Z 739.88,A -85,B 0,C 180,E1 -29148.435,E2 -29148.435} C_VEL
LIN {X 0,Y 54.077,Z 749.869,A -85,B 0,C 180,E1 -29160.003,E2 -29160.003} C_VEL
LIN {X 0,Y 57.827,Z 758.927,A -85,B 0,C 180,E1 -29171.428,E2 -29171.428} C_VEL
LIN {X 0,Y 64.491,Z 767.756,A -85,B 0,C 180,E1 -29182.424,E2 -29182.424} C_VEL
LIN {X 0,Y 74.762,Z 776.158,A -85,B 0,C 180,E1 -29192.222,E2 -29192.222} C_VEL
LIN {X 0,Y 76.488,Z 777.311,A -85,B 0,C 180,E1 -29193.459,E2 -29193.459} C_VEL
LIN {X 0,Y 77.001,Z 777.919,A -85,B 0,C 180,E1 -29194.776,E2 -29194.776} C_VEL
LIN {X 0,Y 68.058,Z 775.097,A -85,B 0,C 180,E1 -29203.715,E2 -29203.715} C_VEL
LIN {X 0,Y 61.82,Z 771.394,A -85,B 0,C 180,E1 -29215.364,E2 -29215.364} C_VEL
LIN {X 0,Y 59.264,Z 766.7,A -85,B 0,C 180,E1 -29229.164,E2 -29229.164} C_VEL
LIN {X 0,Y 60.896,Z 760.771,A -85,B 0,C 180,E1 -29243.377,E2 -29243.377} C_VEL
LIN {X 0,Y 62.32,Z 758.003,A -85,B 0,C 180,E1 -29248.388,E2 -29248.388} C_VEL
LIN {X 0,Y 64.78,Z 752.084,A -85,B 0,C 180,E1 -29256.232,E2 -29256.232} C_VEL
LIN {X 0,Y 65.541,Z 751.16,A -85,B 0,C 180,E1 -29257.648,E2 -29257.648} C_VEL
LIN {X 0,Y 63.748,Z 757.879,A -85,B 0,C 180,E1 -29272.701,E2 -29272.701} C_VEL
LIN {X 0,Y 66.345,Z 762.669,A -85,B 0,C 180,E1 -29285.64,E2 -29285.64} C_VEL
LIN {X 0,Y 73.727,Z 767.132,A -85,B 0,C 180,E1 -29298.14,E2 -29298.14} C_VEL
LIN {X 0,Y 72.255,Z 765.422,A -85,B 0,C 180,E1 -29300.782,E2 -29300.782} C_VEL
LIN {X 0,Y 63.236,Z 754.755,A -85,B 0,C 180,E1 -29311.811,E2 -29311.811} C_VEL
LIN {X 0,Y 58.181,Z 745.054,A -85,B 0,C 180,E1 -29322.42,E2 -29322.42} C_VEL
LIN {X 0,Y 55.249,Z 733.745,A -85,B 0,C 180,E1 -29334.522,E2 -29334.522} C_VEL
LIN {X 0,Y 54.459,Z 723.287,A -85,B 0,C 180,E1 -29344.623,E2 -29344.623} C_VEL
LIN {X 0,Y 55.096,Z 709.595,A -85,B 0,C 180,E1 -29355.724,E2 -29355.724} C_VEL
LIN {X 0,Y 56.814,Z 695.63,A -85,B 0,C 180,E1 -29364.673,E2 -29364.673} C_VEL
LIN {X 0,Y 58.995,Z 681.804,A -85,B 0,C 180,E1 -29371.541,E2 -29371.541} C_VEL
LIN {X 0,Y 61.463,Z 666.452,A -85,B 0,C 180,E1 -29377.193,E2 -29377.193} C_VEL
LIN {X 0,Y 63.884,Z 649.646,A -85,B 0,C 180,E1 -29381.669,E2 -29381.669} C_VEL
LIN {X 0,Y 65.044,Z 639.357,A -85,B 0,C 180,E1 -29384.076,E2 -29384.076} C_VEL
LIN {X 0,Y 62.399,Z 630.842,A -85,B 0,C 180,E1 -29386.455,E2 -29386.455} C_VEL
LIN {X 0,Y 60.387,Z 625.609,A -85,B 0,C 180,E1 -29388.111,E2 -29388.111} C_VEL
LIN {X 0,Y 55.261,Z 617.785,A -85,B 0,C 180,E1 -29391.271,E2 -29391.271} C_VEL
LIN {X 0,Y 48.968,Z 608.494,A -85,B 0,C 180,E1 -29395.929,E2 -29395.929} C_VEL
LIN {X 0,Y 47.47,Z 605.091,A -85,B 0,C 180,E1 -29397.619,E2 -29397.619} C_VEL
LIN {X 0,Y 43.993,Z 595.004,A -85,B 0,C 180,E1 -29402.974,E2 -29402.974} C_VEL
LIN {X 0,Y 44.257,Z 594.969,A -85,B 0,C 180,E1 -29412.313,E2 -29412.313} C_VEL
LIN {X 0,Y 44.55,Z 594.934,A -85,B 0,C 180,E1 -29420.918,E2 -29420.918} C_VEL
LIN {X 0,Y 45.155,Z 594.858,A -85,B 0,C 180,E1 -29429.995,E2 -29429.995} C_VEL
LIN {X 0,Y 44.595,Z 594.927,A -85,B 0,C 180,E1 -29439.062,E2 -29439.062} C_VEL
LIN {X 0,Y 45.711,Z 598.025,A -85,B 0,C 180,E1 -29441.215,E2 -29441.215} C_VEL
LIN {X 0,Y 50.024,Z 608.609,A -85,B 0,C 180,E1 -29447.568,E2 -29447.568} C_VEL
LIN {X 0,Y 54.57,Z 622.457,A -85,B 0,C 180,E1 -29453.732,E2 -29453.732} C_VEL
LIN {X 0,Y 60.058,Z 640.509,A -85,B 0,C 180,E1 -29460.071,E2 -29460.071} C_VEL
LIN {X 0,Y 57.085,Z 664.472,A -85,B 0,C 180,E1 -29464.973,E2 -29464.973} C_VEL
LIN {X 0,Y 54.907,Z 677.493,A -85,B 0,C 180,E1 -29468.379,E2 -29468.379} C_VEL
LIN {X 0,Y 52.2,Z 691.728,A -85,B 0,C 180,E1 -29473.757,E2 -29473.757} C_VEL
LIN {X 0,Y 49.621,Z 704.446,A -85,B 0,C 180,E1 -29480.411,E2 -29480.411} C_VEL
LIN {X 0,Y 47.233,Z 717.68,A -85,B 0,C 180,E1 -29489.86,E2 -29489.86} C_VEL
LIN {X 0,Y 45.949,Z 728.848,A -85,B 0,C 180,E1 -29500.243,E2 -29500.243} C_VEL
LIN {X 0,Y 45.983,Z 738.637,A -85,B 0,C 180,E1 -29511.212,E2 -29511.212} C_VEL
LIN {X 0,Y 48.102,Z 748.779,A -85,B 0,C 180,E1 -29524.193,E2 -29524.193} C_VEL
LIN {X 0,Y 53.039,Z 758.747,A -85,B 0,C 180,E1 -29537.349,E2 -29537.349} C_VEL
LIN {X 0,Y 61.462,Z 768.238,A -85,B 0,C 180,E1 -29549.08,E2 -29549.08} C_VEL
LIN {X 0,Y 66.976,Z 772.785,A -85,B 0,C 180,E1 -29554.068,E2 -29554.068} C_VEL
LIN {X 0,Y 65.594,Z 772.701,A -85,B 0,C 180,E1 -29557.459,E2 -29557.459} C_VEL
LIN {X 0,Y 58.295,Z 769.225,A -85,B 0,C 180,E1 -29568.163,E2 -29568.163} C_VEL
LIN {X 0,Y 53.932,Z 764.471,A -85,B 0,C 180,E1 -29582.874,E2 -29582.874} C_VEL
LIN {X 0,Y 54.172,Z 758.598,A -85,B 0,C 180,E1 -29598.783,E2 -29598.783} C_VEL
LIN {X 0,Y 56.275,Z 754.349,A -85,B 0,C 180,E1 -29607.639,E2 -29607.639} C_VEL
LIN {X 0,Y 59.118,Z 747.861,A -85,B 0,C 180,E1 -29616.832,E2 -29616.832} C_VEL
LIN {X 0,Y 60.012,Z 746.797,A -85,B 0,C 180,E1 -29618.523,E2 -29618.523} C_VEL
LIN {X 0,Y 58.496,Z 753.692,A -85,B 0,C 180,E1 -29634.871,E2 -29634.871} C_VEL
LIN {X 0,Y 63.061,Z 759.754,A -85,B 0,C 180,E1 -29651.971,E2 -29651.971} C_VEL
LIN {X 0,Y 66.5,Z 761.819,A -85,B 0,C 180,E1 -29657.719,E2 -29657.719} C_VEL
LIN {X 0,Y 58.508,Z 752.612,A -85,B 0,C 180,E1 -29667.276,E2 -29667.276} C_VEL
LIN {X 0,Y 52.056,Z 741.032,A -85,B 0,C 180,E1 -29680.271,E2 -29680.271} C_VEL
LIN {X 0,Y 48.854,Z 729.024,A -85,B 0,C 180,E1 -29693.802,E2 -29693.802} C_VEL
LIN {X 0,Y 48.011,Z 717.739,A -85,B 0,C 180,E1 -29705.246,E2 -29705.246} C_VEL
LIN {X 0,Y 48.579,Z 705.548,A -85,B 0,C 180,E1 -29715.735,E2 -29715.735} C_VEL
LIN {X 0,Y 50.157,Z 692.3,A -85,B 0,C 180,E1 -29724.853,E2 -29724.853} C_VEL
LIN {X 0,Y 52.478,Z 678.046,A -85,B 0,C 180,E1 -29732.387,E2 -29732.387} C_VEL
LIN {X 0,Y 55.072,Z 661.525,A -85,B 0,C 180,E1 -29738.677,E2 -29738.677} C_VEL
LIN {X 0,Y 57.825,Z 641.022,A -85,B 0,C 180,E1 -29744.353,E2 -29744.353} C_VEL
LIN {X 0,Y 57.438,Z 638.804,A -85,B 0,C 180,E1 -29745.002,E2 -29745.002} C_VEL
LIN {X 0,Y 47.79,Z 606.096,A -85,B 0,C 180,E1 -29757.155,E2 -29757.155} C_VEL
LIN {X 0,Y 47.47,Z 605.091,A -85,B 0,C 180,E1 -29757.619,E2 -29757.619} C_VEL
LIN {X 0,Y 46.08,Z 603.253,A -85,B 0,C 180,E1 -29758.818,E2 -29758.818} C_VEL
LIN {X 0,Y 38.658,Z 599.47,A -85,B 0,C 180,E1 -29764.192,E2 -29764.192} C_VEL
LIN {X 0,Y 37.542,Z 597.926,A -85,B 0,C 180,E1 -29765.606,E2 -29765.606} C_VEL
LIN {X 0,Y 36.992,Z 595.867,A -85,B 0,C 180,E1 -29767.293,E2 -29767.293} C_VEL
LIN {X 0,Y 37.348,Z 595.832,A -85,B 0,C 180,E1 -29779.147,E2 -29779.147} C_VEL
LIN {X 0,Y 38.014,Z 595.746,A -85,B 0,C 180,E1 -29789.994,E2 -29789.994} C_VEL
LIN {X 0,Y 37.841,Z 595.761,A -85,B 0,C 180,E1 -29791.989,E2 -29791.989} C_VEL
LIN {X 0,Y 38.738,Z 598.686,A -85,B 0,C 180,E1 -29794.546,E2 -29794.546} C_VEL
LIN {X 0,Y 40.093,Z 601.411,A -85,B 0,C 180,E1 -29797.232,E2 -29797.232} C_VEL
LIN {X 0,Y 42.366,Z 607.054,A -85,B 0,C 180,E1 -29801.637,E2 -29801.637} C_VEL
LIN {X 0,Y 46.082,Z 617.784,A -85,B 0,C 180,E1 -29808.041,E2 -29808.041} C_VEL
LIN {X 0,Y 51.606,Z 636.392,A -85,B 0,C 180,E1 -29816.248,E2 -29816.248} C_VEL
LIN {X 0,Y 53.13,Z 641.538,A -85,B 0,C 180,E1 -29818.202,E2 -29818.202} C_VEL
LIN {X 0,Y 50.158,Z 664.169,A -85,B 0,C 180,E1 -29823.357,E2 -29823.357} C_VEL
LIN {X 0,Y 47.712,Z 678.161,A -85,B 0,C 180,E1 -29827.443,E2 -29827.443} C_VEL
LIN {X 0,Y 44.926,Z 692.391,A -85,B 0,C 180,E1 -29833.661,E2 -29833.661} C_VEL
LIN {X 0,Y 41.974,Z 706.658,A -85,B 0,C 180,E1 -29842.636,E2 -29842.636} C_VEL
LIN {X 0,Y 39.915,Z 719.346,A -85,B 0,C 180,E1 -29853.661,E2 -29853.661} C_VEL
LIN {X 0,Y 39.213,Z 731.098,A -85,B 0,C 180,E1 -29867.059,E2 -29867.059} C_VEL
LIN {X 0,Y 40.778,Z 742.54,A -85,B 0,C 180,E1 -29882.474,E2 -29882.474} C_VEL
LIN {X 0,Y 44.902,Z 752.451,A -85,B 0,C 180,E1 -29896.394,E2 -29896.394} C_VEL
LIN {X 0,Y 52.959,Z 762.896,A -85,B 0,C 180,E1 -29909.848,E2 -29909.848} C_VEL
LIN {X 0,Y 58.014,Z 767.564,A -85,B 0,C 180,E1 -29915.134,E2 -29915.134} C_VEL
LIN {X 0,Y 57.877,Z 767.876,A -85,B 0,C 180,E1 -29917.387,E2 -29917.387} C_VEL
LIN {X 0,Y 50.606,Z 763.332,A -85,B 0,C 180,E1 -29931.328,E2 -29931.328} C_VEL
LIN {X 0,Y 47.867,Z 757.408,A -85,B 0,C 180,E1 -29949.78,E2 -29949.78} C_VEL
LIN {X 0,Y 50.129,Z 751.001,A -85,B 0,C 180,E1 -29965.865,E2 -29965.865} C_VEL
LIN {X 0,Y 52.614,Z 744.883,A -85,B 0,C 180,E1 -29975.418,E2 -29975.418} C_VEL
LIN {X 0,Y 54.684,Z 742.22,A -85,B 0,C 180,E1 -29979.361,E2 -29979.361} C_VEL
LIN {X 0,Y 53.227,Z 747.896,A -85,B 0,C 180,E1 -29993.34,E2 -29993.34} C_VEL
LIN {X 0,Y 55.918,Z 753.313,A -85,B 0,C 180,E1 -30008.939,E2 -30008.939} C_VEL
LIN {X 0,Y 58.862,Z 755.659,A -85,B 0,C 180,E1 -30015.763,E2 -30015.763} C_VEL
LIN {X 0,Y 57.858,Z 754.456,A -85,B 0,C 180,E1 -30017.608,E2 -30017.608} C_VEL
LIN {X 0,Y 50.225,Z 744.491,A -85,B 0,C 180,E1 -30028.345,E2 -30028.345} C_VEL
LIN {X 0,Y 44.851,Z 733.197,A -85,B 0,C 180,E1 -30041.732,E2 -30041.732} C_VEL
LIN {X 0,Y 42.318,Z 721.802,A -85,B 0,C 180,E1 -30055.237,E2 -30055.237} C_VEL
LIN {X 0,Y 41.712,Z 709.175,A -85,B 0,C 180,E1 -30068.473,E2 -30068.473} C_VEL
LIN {X 0,Y 42.79,Z 695.216,A -85,B 0,C 180,E1 -30080.423,E2 -30080.423} C_VEL
LIN {X 0,Y 44.747,Z 681.553,A -85,B 0,C 180,E1 -30089.39,E2 -30089.39} C_VEL
LIN {X 0,Y 47.1,Z 666.529,A -85,B 0,C 180,E1 -30096.641,E2 -30096.641} C_VEL
LIN {X 0,Y 49.879,Z 647.815,A -85,B 0,C 180,E1 -30103.007,E2 -30103.007} C_VEL
LIN {X 0,Y 50.724,Z 641.118,A -85,B 0,C 180,E1 -30105.031,E2 -30105.031} C_VEL
LIN {X 0,Y 41.413,Z 609.002,A -85,B 0,C 180,E1 -30118.68,E2 -30118.68} C_VEL
LIN {X 0,Y 37.765,Z 598.387,A -85,B 0,C 180,E1 -30125.242,E2 -30125.242} C_VEL
LIN {X 0,Y 37.542,Z 597.926,A -85,B 0,C 180,E1 -30125.606,E2 -30125.606} C_VEL
LIN {X 0,Y 36.838,Z 596.814,A -85,B 0,C 180,E1 -30127.581,E2 -30127.581} C_VEL
LIN {X 0,Y 35.83,Z 596.59,A -85,B 0,C 180,E1 -30132.288,E2 -30132.288} C_VEL
LIN {X 0,Y 35.307,Z 597.544,A -85,B 0,C 180,E1 -30136.997,E2 -30136.997} C_VEL
LIN {X 0,Y 35.191,Z 600.044,A -85,B 0,C 180,E1 -30143.526,E2 -30143.526} C_VEL
LIN {X 0,Y 35.825,Z 604.331,A -85,B 0,C 180,E1 -30150.236,E2 -30150.236} C_VEL
LIN {X 0,Y 37.234,Z 610.322,A -85,B 0,C 180,E1 -30157.187,E2 -30157.187} C_VEL
LIN {X 0,Y 38.908,Z 616.872,A -85,B 0,C 180,E1 -30162.342,E2 -30162.342} C_VEL
LIN {X 0,Y 43.266,Z 631.961,A -85,B 0,C 180,E1 -30171.041,E2 -30171.041} C_VEL
LIN {X 0,Y 46.226,Z 642.788,A -85,B 0,C 180,E1 -30175.949,E2 -30175.949} C_VEL
LIN {X 0,Y 42.996,Z 665.477,A -85,B 0,C 180,E1 -30181.919,E2 -30181.919} C_VEL
LIN {X 0,Y 40.188,Z 680.425,A -85,B 0,C 180,E1 -30187.079,E2 -30187.079} C_VEL
LIN {X 0,Y 37.172,Z 694.913,A -85,B 0,C 180,E1 -30194.854,E2 -30194.854} C_VEL
LIN {X 0,Y 34.469,Z 708.281,A -85,B 0,C 180,E1 -30205.394,E2 -30205.394} C_VEL
LIN {X 0,Y 32.801,Z 721.089,A -85,B 0,C 180,E1 -30219.63,E2 -30219.63} C_VEL
LIN {X 0,Y 33.241,Z 733.425,A -85,B 0,C 180,E1 -30236.976,E2 -30236.976} C_VEL
LIN {X 0,Y 36.415,Z 744.116,A -85,B 0,C 180,E1 -30253.408,E2 -30253.408} C_VEL
LIN {X 0,Y 43.409,Z 755.228,A -85,B 0,C 180,E1 -30269.064,E2 -30269.064} C_VEL
LIN {X 0,Y 49.853,Z 761.978,A -85,B 0,C 180,E1 -30277.063,E2 -30277.063} C_VEL
LIN {X 0,Y 48.852,Z 761.585,A -85,B 0,C 180,E1 -30280.302,E2 -30280.302} C_VEL
LIN {X 0,Y 43.43,Z 756.587,A -85,B 0,C 180,E1 -30296.505,E2 -30296.505} C_VEL
LIN {X 0,Y 42.673,Z 750.962,A -85,B 0,C 180,E1 -30314.357,E2 -30314.357} C_VEL
LIN {X 0,Y 44.462,Z 746.673,A -85,B 0,C 180,E1 -30325.278,E2 -30325.278} C_VEL
LIN {X 0,Y 47.249,Z 740.136,A -85,B 0,C 180,E1 -30336.41,E2 -30336.41} C_VEL
LIN {X 0,Y 49.463,Z 737.559,A -85,B 0,C 180,E1 -30340.494,E2 -30340.494} C_VEL
LIN {X 0,Y 48.584,Z 744.651,A -85,B 0,C 180,E1 -30359.772,E2 -30359.772} C_VEL
LIN {X 0,Y 51.674,Z 748.942,A -85,B 0,C 180,E1 -30372.852,E2 -30372.852} C_VEL
LIN {X 0,Y 50.619,Z 747.593,A -85,B 0,C 180,E1 -30376.032,E2 -30376.032} C_VEL
LIN {X 0,Y 43.028,Z 736.86,A -85,B 0,C 180,E1 -30387.933,E2 -30387.933} C_VEL
LIN {X 0,Y 38.357,Z 726.203,A -85,B 0,C 180,E1 -30401.293,E2 -30401.293} C_VEL
LIN {X 0,Y 36.093,Z 715.858,A -85,B 0,C 180,E1 -30414.408,E2 -30414.408} C_VEL
LIN {X 0,Y 35.5,Z 701.868,A -85,B 0,C 180,E1 -30430.113,E2 -30430.113} C_VEL
LIN {X 0,Y 36.485,Z 689.83,A -85,B 0,C 180,E1 -30441.167,E2 -30441.167} C_VEL
LIN {X 0,Y 38.631,Z 674.938,A -85,B 0,C 180,E1 -30451.531,E2 -30451.531} C_VEL
LIN {X 0,Y 41.064,Z 659.337,A -85,B 0,C 180,E1 -30459.126,E2 -30459.126} C_VEL
LIN {X 0,Y 43.578,Z 641.992,A -85,B 0,C 180,E1 -30465.524,E2 -30465.524} C_VEL
LIN {X 0,Y 34.887,Z 611.307,A -85,B 0,C 180,E1 -30480.997,E2 -30480.997} C_VEL
LIN {X 0,Y 31.769,Z 601.779,A -85,B 0,C 180,E1 -30488.223,E2 -30488.223} C_VEL
LIN {X 0,Y 30.057,Z 596.62,A -85,B 0,C 180,E1 -30493.162,E2 -30493.162} C_VEL
LIN {X 0,Y 30.271,Z 596.682,A -85,B 0,C 180,E1 -30499.119,E2 -30499.119} C_VEL
LIN {X 0,Y 31.232,Z 599.273,A -85,B 0,C 180,E1 -30503.126,E2 -30503.126} C_VEL
LIN {X 0,Y 33.193,Z 601.337,A -85,B 0,C 180,E1 -30508.097,E2 -30508.097} C_VEL
LIN {X 0,Y 36.038,Z 608.164,A -85,B 0,C 180,E1 -30515.607,E2 -30515.607} C_VEL
LIN {X 0,Y 38.908,Z 616.872,A -85,B 0,C 180,E1 -30522.342,E2 -30522.342} C_VEL
LIN {X 0,Y 39.26,Z 620.642,A -85,B 0,C 180,E1 -30524.143,E2 -30524.143} C_VEL
LIN {X 0,Y 38.369,Z 627.198,A -85,B 0,C 180,E1 -30525.987,E2 -30525.987} C_VEL
LIN {X 0,Y 37.426,Z 633.771,A -85,B 0,C 180,E1 -30527.88,E2 -30527.88} C_VEL
LIN {X 0,Y 37.793,Z 637.573,A -85,B 0,C 180,E1 -30529.655,E2 -30529.655} C_VEL
LIN {X 0,Y 39.366,Z 644.176,A -85,B 0,C 180,E1 -30533.132,E2 -30533.132} C_VEL
LIN {X 0,Y 35.616,Z 667.919,A -85,B 0,C 180,E1 -30540.32,E2 -30540.32} C_VEL
LIN {X 0,Y 32.628,Z 682.643,A -85,B 0,C 180,E1 -30546.653,E2 -30546.653} C_VEL
LIN {X 0,Y 29.573,Z 696.703,A -85,B 0,C 180,E1 -30556.37,E2 -30556.37} C_VEL
LIN {X 0,Y 26.981,Z 710.436,A -85,B 0,C 180,E1 -30570.772,E2 -30570.772} C_VEL
LIN {X 0,Y 26.142,Z 721.278,A -85,B 0,C 180,E1 -30586.401,E2 -30586.401} C_VEL
LIN {X 0,Y 27.729,Z 732.781,A -85,B 0,C 180,E1 -30606.008,E2 -30606.008} C_VEL
LIN {X 0,Y 33.034,Z 744.508,A -85,B 0,C 180,E1 -30625.188,E2 -30625.188} C_VEL
LIN {X 0,Y 40.257,Z 753.801,A -85,B 0,C 180,E1 -30637.67,E2 -30637.67} C_VEL
LIN {X 0,Y 42.052,Z 755.685,A -85,B 0,C 180,E1 -30639.827,E2 -30639.827} C_VEL
LIN {X 0,Y 41.146,Z 755.047,A -85,B 0,C 180,E1 -30643.102,E2 -30643.102} C_VEL
LIN {X 0,Y 37.324,Z 749.657,A -85,B 0,C 180,E1 -30661.925,E2 -30661.925} C_VEL
LIN {X 0,Y 38.462,Z 743.293,A -85,B 0,C 180,E1 -30682.016,E2 -30682.016} C_VEL
LIN {X 0,Y 41.23,Z 736.422,A -85,B 0,C 180,E1 -30695.385,E2 -30695.385} C_VEL
LIN {X 0,Y 44.38,Z 732.729,A -85,B 0,C 180,E1 -30701.999,E2 -30701.999} C_VEL
LIN {X 0,Y 43.574,Z 738.624,A -85,B 0,C 180,E1 -30718.944,E2 -30718.944} C_VEL
LIN {X 0,Y 45.061,Z 741.662,A -85,B 0,C 180,E1 -30728.749,E2 -30728.749} C_VEL
LIN {X 0,Y 45.46,Z 742.188,A -85,B 0,C 180,E1 -30731.725,E2 -30731.725} C_VEL
LIN {X 0,Y 36.968,Z 730.134,A -85,B 0,C 180,E1 -30745.221,E2 -30745.221} C_VEL
LIN {X 0,Y 31.915,Z 718.215,A -85,B 0,C 180,E1 -30761.11,E2 -30761.11} C_VEL
LIN {X 0,Y 29.602,Z 706.063,A -85,B 0,C 180,E1 -30777.442,E2 -30777.442} C_VEL
LIN {X 0,Y 29.531,Z 692.397,A -85,B 0,C 180,E1 -30793.762,E2 -30793.762} C_VEL
LIN {X 0,Y 31.165,Z 677.111,A -85,B 0,C 180,E1 -30807.711,E2 -30807.711} C_VEL
LIN {X 0,Y 33.332,Z 662.804,A -85,B 0,C 180,E1 -30816.835,E2 -30816.835} C_VEL
LIN {X 0,Y 36.312,Z 642.974,A -85,B 0,C 180,E1 -30826.022,E2 -30826.022} C_VEL
LIN {X 0,Y 30.317,Z 621.299,A -85,B 0,C 180,E1 -30838.552,E2 -30838.552} C_VEL
LIN {X 0,Y 27.64,Z 610.946,A -85,B 0,C 180,E1 -30846.5,E2 -30846.5} C_VEL
LIN {X 0,Y 25.771,Z 604.849,A -85,B 0,C 180,E1 -30852.611,E2 -30852.611} C_VEL
LIN {X 0,Y 27.542,Z 604.79,A -85,B 0,C 180,E1 -30858.204,E2 -30858.204} C_VEL
LIN {X 0,Y 29.124,Z 607.077,A -85,B 0,C 180,E1 -30863.801,E2 -30863.801} C_VEL
LIN {X 0,Y 30.947,Z 612.158,A -85,B 0,C 180,E1 -30870.531,E2 -30870.531} C_VEL
LIN {X 0,Y 33.521,Z 621.305,A -85,B 0,C 180,E1 -30878.875,E2 -30878.875} C_VEL
LIN {X 0,Y 37.252,Z 635.429,A -85,B 0,C 180,E1 -30888.419,E2 -30888.419} C_VEL
LIN {X 0,Y 37.793,Z 637.573,A -85,B 0,C 180,E1 -30889.655,E2 -30889.655} C_VEL
LIN {X 0,Y 37.902,Z 640.649,A -85,B 0,C 180,E1 -30890.918,E2 -30890.918} C_VEL
LIN {X 0,Y 36.5,Z 644.994,A -85,B 0,C 180,E1 -30891.713,E2 -30891.713} C_VEL
LIN {X 0,Y 31.292,Z 654.827,A -85,B 0,C 180,E1 -30892.591,E2 -30892.591} C_VEL
LIN {X 0,Y 30.552,Z 657.484,A -85,B 0,C 180,E1 -30893.35,E2 -30893.35} C_VEL
LIN {X 0,Y 27.437,Z 673.719,A -85,B 0,C 180,E1 -30899.767,E2 -30899.767} C_VEL
LIN {X 0,Y 24.329,Z 687.759,A -85,B 0,C 180,E1 -30908.563,E2 -30908.563} C_VEL
LIN {X 0,Y 21.444,Z 700.896,A -85,B 0,C 180,E1 -30922.094,E2 -30922.094} C_VEL
LIN {X 0,Y 19.879,Z 713.399,A -85,B 0,C 180,E1 -30941.989,E2 -30941.989} C_VEL
LIN {X 0,Y 21.277,Z 726.287,A -85,B 0,C 180,E1 -30967.808,E2 -30967.808} C_VEL
LIN {X 0,Y 26.425,Z 737.924,A -85,B 0,C 180,E1 -30989.102,E2 -30989.102} C_VEL
LIN {X 0,Y 34.472,Z 748.391,A -85,B 0,C 180,E1 -31003.319,E2 -31003.319} C_VEL
LIN {X 0,Y 33.357,Z 747.015,A -85,B 0,C 180,E1 -31010.806,E2 -31010.806} C_VEL
LIN {X 0,Y 32.738,Z 739.701,A -85,B 0,C 180,E1 -31037.611,E2 -31037.611} C_VEL
LIN {X 0,Y 33.783,Z 735.854,A -85,B 0,C 180,E1 -31047.133,E2 -31047.133} C_VEL
LIN {X 0,Y 36.716,Z 730.583,A -85,B 0,C 180,E1 -31057.984,E2 -31057.984} C_VEL
LIN {X 0,Y 39.527,Z 727.662,A -85,B 0,C 180,E1 -31063.459,E2 -31063.459} C_VEL
LIN {X 0,Y 39.143,Z 733.746,A -85,B 0,C 180,E1 -31082.598,E2 -31082.598} C_VEL
LIN {X 0,Y 38.891,Z 734.045,A -85,B 0,C 180,E1 -31088.55,E2 -31088.55} C_VEL
LIN {X 0,Y 31.138,Z 722.644,A -85,B 0,C 180,E1 -31101.626,E2 -31101.626} C_VEL
LIN {X 0,Y 26.414,Z 711.937,A -85,B 0,C 180,E1 -31116.47,E2 -31116.47} C_VEL
LIN {X 0,Y 23.641,Z 699.005,A -85,B 0,C 180,E1 -31135.73,E2 -31135.73} C_VEL
LIN {X 0,Y 23.455,Z 685.167,A -85,B 0,C 180,E1 -31154.497,E2 -31154.497} C_VEL
LIN {X 0,Y 24.902,Z 671.826,A -85,B 0,C 180,E1 -31168.375,E2 -31168.375} C_VEL
LIN {X 0,Y 27.966,Z 651.364,A -85,B 0,C 180,E1 -31182.422,E2 -31182.422} C_VEL
LIN {X 0,Y 29.018,Z 642.96,A -85,B 0,C 180,E1 -31187.103,E2 -31187.103} C_VEL
LIN {X 0,Y 22.043,Z 615.98,A -85,B 0,C 180,E1 -31208.987,E2 -31208.987} C_VEL
LIN {X 0,Y 22.314,Z 615.779,A -85,B 0,C 180,E1 -31210.862,E2 -31210.862} C_VEL
LIN {X 0,Y 23.928,Z 615.195,A -85,B 0,C 180,E1 -31216.382,E2 -31216.382} C_VEL
LIN {X 0,Y 25.363,Z 613.931,A -85,B 0,C 180,E1 -31219.646,E2 -31219.646} C_VEL
LIN {X 0,Y 25.739,Z 614.206,A -85,B 0,C 180,E1 -31220.909,E2 -31220.909} C_VEL
LIN {X 0,Y 27.661,Z 622.812,A -85,B 0,C 180,E1 -31231.347,E2 -31231.347} C_VEL
LIN {X 0,Y 30.82,Z 636.853,A -85,B 0,C 180,E1 -31243.594,E2 -31243.594} C_VEL
LIN {X 0,Y 32.674,Z 644.707,A -85,B 0,C 180,E1 -31248.971,E2 -31248.971} C_VEL
LIN {X 0,Y 30.552,Z 657.484,A -85,B 0,C 180,E1 -31253.35,E2 -31253.35} C_VEL
LIN {X 0,Y 28.915,Z 663.092,A -85,B 0,C 180,E1 -31254.993,E2 -31254.993} C_VEL
LIN {X 0,Y 24.344,Z 671.862,A -85,B 0,C 180,E1 -31256.861,E2 -31256.861} C_VEL
LIN {X 0,Y 19.509,Z 680.507,A -85,B 0,C 180,E1 -31260.261,E2 -31260.261} C_VEL
LIN {X 0,Y 17.568,Z 685.935,A -85,B 0,C 180,E1 -31264.817,E2 -31264.817} C_VEL
LIN {X 0,Y 14.614,Z 698.917,A -85,B 0,C 180,E1 -31283.064,E2 -31283.064} C_VEL
LIN {X 0,Y 13.814,Z 713.281,A -85,B 0,C 180,E1 -31316.367,E2 -31316.367} C_VEL
LIN {X 0,Y 17.649,Z 725.881,A -85,B 0,C 180,E1 -31346.835,E2 -31346.835} C_VEL
LIN {X 0,Y 26.318,Z 738.879,A -85,B 0,C 180,E1 -31367.264,E2 -31367.264} C_VEL
LIN {X 0,Y 27.825,Z 740.688,A -85,B 0,C 180,E1 -31369.275,E2 -31369.275} C_VEL
LIN {X 0,Y 27.287,Z 738.979,A -85,B 0,C 180,E1 -31379.006,E2 -31379.006} C_VEL
LIN {X 0,Y 27.591,Z 734.933,A -85,B 0,C 180,E1 -31395.252,E2 -31395.252} C_VEL
LIN {X 0,Y 30.027,Z 727.804,A -85,B 0,C 180,E1 -31414.149,E2 -31414.149} C_VEL
LIN {X 0,Y 34.881,Z 722.441,A -85,B 0,C 180,E1 -31425.292,E2 -31425.292} C_VEL
LIN {X 0,Y 34.256,Z 725.119,A -85,B 0,C 180,E1 -31434.233,E2 -31434.233} C_VEL
LIN {X 0,Y 33.637,Z 726.25,A -85,B 0,C 180,E1 -31443.296,E2 -31443.296} C_VEL
LIN {X 0,Y 26.2,Z 715.386,A -85,B 0,C 180,E1 -31455.231,E2 -31455.231} C_VEL
LIN {X 0,Y 20.647,Z 703.414,A -85,B 0,C 180,E1 -31472.083,E2 -31472.083} C_VEL
LIN {X 0,Y 17.708,Z 690.285,A -85,B 0,C 180,E1 -31494.295,E2 -31494.295} C_VEL
LIN {X 0,Y 17.627,Z 675.682,A -85,B 0,C 180,E1 -31517.388,E2 -31517.388} C_VEL
LIN {X 0,Y 19.499,Z 659.619,A -85,B 0,C 180,E1 -31535.25,E2 -31535.25} C_VEL
LIN {X 0,Y 21.833,Z 644.533,A -85,B 0,C 180,E1 -31547.337,E2 -31547.337} C_VEL
LIN {X 0,Y 21.041,Z 640.737,A -85,B 0,C 180,E1 -31550.439,E2 -31550.439} C_VEL
LIN {X 0,Y 17.758,Z 628.208,A -85,B 0,C 180,E1 -31563.546,E2 -31563.546} C_VEL
LIN {X 0,Y 18.56,Z 628.167,A -85,B 0,C 180,E1 -31568.761,E2 -31568.761} C_VEL
LIN {X 0,Y 20.571,Z 626.508,A -85,B 0,C 180,E1 -31576.072,E2 -31576.072} C_VEL
LIN {X 0,Y 21.527,Z 625.329,A -85,B 0,C 180,E1 -31578.311,E2 -31578.311} C_VEL
LIN {X 0,Y 22.58,Z 625.364,A -85,B 0,C 180,E1 -31581.671,E2 -31581.671} C_VEL
LIN {X 0,Y 25.123,Z 640.594,A -85,B 0,C 180,E1 -31598.623,E2 -31598.623} C_VEL
LIN {X 0,Y 26.069,Z 646.202,A -85,B 0,C 180,E1 -31603.398,E2 -31603.398} C_VEL
LIN {X 0,Y 21.641,Z 668.889,A -85,B 0,C 180,E1 -31612.843,E2 -31612.843} C_VEL
LIN {X 0,Y 18.183,Z 683.407,A -85,B 0,C 180,E1 -31622.318,E2 -31622.318} C_VEL
LIN {X 0,Y 17.568,Z 685.935,A -85,B 0,C 180,E1 -31624.817,E2 -31624.817} C_VEL
LIN {X 0,Y 15.67,Z 691.231,A -85,B 0,C 180,E1 -31630.89,E2 -31630.89} C_VEL
LIN {X 0,Y 12.997,Z 696.131,A -85,B 0,C 180,E1 -31639.045,E2 -31639.045} C_VEL
LIN {X 0,Y 8.505,Z 705.379,A -85,B 0,C 180,E1 -31673.392,E2 -31673.392} C_VEL
LIN {X 0,Y 8.74,Z 710.161,A -85,B 0,C 180,E1 -31697.494,E2 -31697.494} C_VEL
LIN {X 0,Y 9.302,Z 711.823,A -85,B 0,C 180,E1 -31703.578,E2 -31703.578} C_VEL
LIN {X 0,Y 16.067,Z 724.254,A -85,B 0,C 180,E1 -31729.969,E2 -31729.969} C_VEL
LIN {X 0,Y 21.814,Z 731.926,A -85,B 0,C 180,E1 -31738.44,E2 -31738.44} C_VEL
LIN {X 0,Y 22.523,Z 730.599,A -85,B 0,C 180,E1 -31749.43,E2 -31749.43} C_VEL
LIN {X 0,Y 25.101,Z 722.505,A -85,B 0,C 180,E1 -31774.965,E2 -31774.965} C_VEL
LIN {X 0,Y 30.321,Z 717.159,A -85,B 0,C 180,E1 -31787.498,E2 -31787.498} C_VEL
LIN {X 0,Y 30.135,Z 718.044,A -85,B 0,C 180,E1 -31791.095,E2 -31791.095} C_VEL
LIN {X 0,Y 29.59,Z 718.586,A -85,B 0,C 180,E1 -31795.661,E2 -31795.661} C_VEL
LIN {X 0,Y 21.787,Z 707.202,A -85,B 0,C 180,E1 -31806.235,E2 -31806.235} C_VEL
LIN {X 0,Y 15.211,Z 693.569,A -85,B 0,C 180,E1 -31824.708,E2 -31824.708} C_VEL
LIN {X 0,Y 11.923,Z 680.02,A -85,B 0,C 180,E1 -31851.51,E2 -31851.51} C_VEL
LIN {X 0,Y 11.96,Z 664.373,A -85,B 0,C 180,E1 -31882.666,E2 -31882.666} C_VEL
LIN {X 0,Y 14.692,Z 644.412,A -85,B 0,C 180,E1 -31909.171,E2 -31909.171} C_VEL
LIN {X 0,Y 13.707,Z 640.889,A -85,B 0,C 180,E1 -31914.188,E2 -31914.188} C_VEL
LIN {X 0,Y 14.533,Z 640.77,A -85,B 0,C 180,E1 -31923.802,E2 -31923.802} C_VEL
LIN {X 0,Y 16.327,Z 638.846,A -85,B 0,C 180,E1 -31932.777,E2 -31932.777} C_VEL
LIN {X 0,Y 18.693,Z 635.478,A -85,B 0,C 180,E1 -31939.141,E2 -31939.141} C_VEL
LIN {X 0,Y 20.001,Z 646.753,A -85,B 0,C 180,E1 -31953.972,E2 -31953.972} C_VEL
LIN {X 0,Y 15.073,Z 668.456,A -85,B 0,C 180,E1 -31963.983,E2 -31963.983} C_VEL
LIN {X 0,Y 10.902,Z 684.185,A -85,B 0,C 180,E1 -31977.611,E2 -31977.611} C_VEL
LIN {X 0,Y 7.918,Z 696.362,A -85,B 0,C 180,E1 -32004.402,E2 -32004.402} C_VEL
LIN {X 0,Y 8.446,Z 709.305,A -85,B 0,C 180,E1 -32054.879,E2 -32054.879} C_VEL
LIN {X 0,Y 9.302,Z 711.823,A -85,B 0,C 180,E1 -32063.578,E2 -32063.578} C_VEL
LIN {X 0,Y 10.079,Z 714.016,A -85,B 0,C 180,E1 -32073.562,E2 -32073.562} C_VEL
LIN {X 0,Y 10.908,Z 715.708,A -85,B 0,C 180,E1 -32085.707,E2 -32085.707} C_VEL
LIN {X 0,Y 12.759,Z 717.407,A -85,B 0,C 180,E1 -32103.919,E2 -32103.919} C_VEL
LIN {X 0,Y 15.38,Z 718.136,A -85,B 0,C 180,E1 -32118.898,E2 -32118.898} C_VEL
LIN {X 0,Y 18.674,Z 717.734,A -85,B 0,C 180,E1 -32131.1,E2 -32131.1} C_VEL
LIN {X 0,Y 20.954,Z 716.298,A -85,B 0,C 180,E1 -32138.398,E2 -32138.398} C_VEL
LIN {X 0,Y 21.144,Z 716.088,A -85,B 0,C 180,E1 -32139.047,E2 -32139.047} C_VEL
LIN {X 0,Y 22.585,Z 714.53,A -85,B 0,C 180,E1 -32143.471,E2 -32143.471} C_VEL
LIN {X 0,Y 21.884,Z 712.559,A -85,B 0,C 180,E1 -32145.507,E2 -32145.507} C_VEL
LIN {X 0,Y 11.914,Z 698.081,A -85,B 0,C 180,E1 -32157.74,E2 -32157.74} C_VEL
LIN {X 0,Y 6.042,Z 686.127,A -85,B 0,C 180,E1 -32186.926,E2 -32186.926} C_VEL
LIN {X 0,Y 5.974,Z 671.14,A -85,B 0,C 180,E1 -32261.799,E2 -32261.799} C_VEL
LIN {X 0,Y 14.491,Z 647.179,A -85,B 0,C 180,E1 -32295.873,E2 -32295.873} C_VEL
LIN {X 0,Y 14.677,Z 647.694,A -85,B 0,C 180,E1 -32297.682,E2 -32297.682} C_VEL
LIN {X 0,Y 9.506,Z 667.417,A -85,B 0,C 180,E1 -32303.293,E2 -32303.293} C_VEL
LIN {X 0,Y 4.608,Z 683.124,A -85,B 0,C 180,E1 -32312.666,E2 -32312.666} C_VEL
LIN {X 0,Y 1.71,Z 695.787,A -85,B 0,C 180,E1 -32422.41,E2 -32422.41} C_VEL
LIN {X 0,Y 8.667,Z 709.701,A -85,B 0,C 180,E1 -32467.612,E2 -32467.612} C_VEL
LIN {X 0,Y 17.413,Z 722.57,A -85,B 0,C 180,E1 -32473.485,E2 -32473.485} C_VEL
LIN {X 0,Y 17.987,Z 721.788,A -85,B 0,C 180,E1 -32478.736,E2 -32478.736} C_VEL
LIN {X 0,Y 21.144,Z 716.088,A -85,B 0,C 180,E1 -32499.047,E2 -32499.047} C_VEL
LIN {X 0,Y 21.144,Z 716.088,A -85,B 0,C 180,E1 -32499.047,E2 -32499.047}

QRS_NEXT_CUT()

QRS_NEXT()
QRS_HOME()

END
